{attribute 'linkalways'} 
{attribute 'no_explicit_call' := 'This FB is a CLASS and must be accessed using methods or properties'}
{attribute 'enable_dynamic_creation'}
FUNCTION_BLOCK _TcVnVector3_INT EXTENDS AliasDatatypeBase
VAR
	localData : TcVnVector3_INT;
	activeData : REFERENCE TO TcVnVector3_INT REF= localData;
	aliasBaseDatatype : _Array0to2OfINT;
END_VAR

PROPERTY PUBLIC Address : PVOID
GET
Address := ADR(activeData);
END_GET
END_PROPERTY

METHOD PUBLIC ClearReference
VAR_INPUT
END_VAR
activeData REF= localData;
SetBaseDatatypeReference();
END_METHOD

METHOD PUBLIC Clone : I_Datatype
VAR
    pClone : POINTER TO _TcVnVector3_INT;
END_VAR
pClone := __NEW(_TcVnVector3_INT);
Clone := pClone^;
END_METHOD

METHOD FB_init : BOOL
VAR_INPUT
	bInitRetains : BOOL; // if TRUE, the retain variables are initialized (warm start / cold start)
	bInCopyCode : BOOL;  // if TRUE, the instance afterwards gets moved into the copy code (online change)
	//InitialValue : <type>; // if possible, not all values can be initialized
END_VAR
//localData := InitialValue; // if possible, not all values can be initialized
SetBaseDatatypeReference();
AddBaseDatatype(aliasBaseDatatype);
END_METHOD

PROPERTY PUBLIC Identifier : T_MAXSTRING
GET
Identifier := 'TcVnVector3_INT';
END_GET
END_PROPERTY

METHOD PUBLIC MakeReferenceTo
VAR_INPUT
	ReferenceTarget : REFERENCE TO TcVnVector3_INT;
END_VAR
activeData REF= ReferenceTarget;
SetBaseDatatypeReference();
END_METHOD

METHOD PROTECTED SetBaseDatatypeReference
VAR_INPUT
END_VAR
aliasBaseDatatype.MakeReferenceTo(activeData);
END_METHOD

PROPERTY PUBLIC Size : UDINT
GET
Size := SIZEOF(activeData);
END_GET
END_PROPERTY

METHOD TryMakeReferenceTo : BOOL
VAR_INPUT
	Target : I_Datatype;
END_VAR
VAR
	pTargetData : POINTER TO TcVnVector3_INT;
END_VAR
IF NOT IsEquivalentTo(Target) THEN
	RETURN;
END_IF

pTargetData := Target.Address;
activeData REF= pTargetData^;
SetBaseDatatypeReference();
TryMakeReferenceTo := TRUE;
END_METHOD

PROPERTY PUBLIC Value : REFERENCE TO TcVnVector3_INT
GET
Value REF= activeData;
END_GET
END_PROPERTY

END_FUNCTION_BLOCK

(* stored: Version 1.1.0.1, ProductVersion 3.1.4024.13
   POU _TcVnVector3_INT: Id {8492fb69-2f1a-09de-3605-979f3e6ad7da}, SpecialFunc None
   Folder Core: Id {16bb31e0-deeb-0366-02e7-7f80bc159c9c}
   Folder Protected: Id {405b6a65-436e-0230-2bc6-cf13ba736384}
   Folder Customize: Id {4ee0bb70-2612-0a9e-3a59-a33acf37ef87}
   Folder Constructor: Id {63372253-55da-028e-1583-6bc89ea9fe60}
   Property Address: Id {533b66e7-799c-03e8-2920-4302daff0ce0}
   Get Get: Id {2e9b44c2-6cd3-090f-008d-935803c0d40a}
   Method ClearReference: Id {d5dba117-6e64-0de2-1447-15fdc2de12c2}
   Method Clone: Id {1b2d08b8-9b05-0c0f-3a9c-ec907e3b9be1}
   Method FB_init: Id {d14611b1-899e-0f99-2d81-7cfdb03ee12c}
   Property Identifier: Id {e5a2d062-f7a7-097f-26a8-a8b49b9f93da}
   Get Get: Id {fbc921f5-8f10-08bd-08b2-2800d022f0fd}
   Method MakeReferenceTo: Id {31010d56-0e20-0cbf-003c-2ed03b1fca18}
   Method SetBaseDatatypeReference: Id {3af67e29-6ad0-00db-0048-e2e00aff34fb}
   Property Size: Id {3efb12fb-04f5-0416-12a8-1baee4fcae12}
   Get Get: Id {a671335d-a7c9-09aa-2ebf-b714c3691883}
   Method TryMakeReferenceTo: Id {039e36d5-e696-0656-29d2-21cd93956591}
   Property Value: Id {db84b1fd-51cc-07f0-1a33-fd4136317beb}
   Get Get: Id {63ff0400-c49d-0686-334d-cd3043934140} *)
